{attribute 'qualified_only'}
{attribute 'strict'}
{attribute 'to_string'}
{info 'E_APP_VARIANT placeholder for application variant; add new members here'}
TYPE E_APP_VARIANT :
(
  VARIANT_INVALID
);
END_TYPE

(* stored: Version 1.1.0.1, ProductVersion 3.1.4026.18
   DUT E_APP_VARIANT: Id {cf52a74b-c1c1-4fa1-922c-ea41bc632144} *)
